{attribute 'linkalways'} 
{attribute 'no_explicit_call' := 'This FB is a CLASS and must be accessed using methods or properties'}
{attribute 'enable_dynamic_creation'}
FUNCTION_BLOCK Node_F_VN_BitwiseAndImages EXTENDS VisionNode
VAR
    ipSrcImage1 : _ITcVnImage;
    ipSrcImage2 : _ITcVnImage;
    ipDestImage : _ITcVnImage;
    hrPrev : _HRESULT(S_OK);
	hresult : _HRESULT(S_OK);
END_VAR

METHOD PUBLIC  Clone : I_Node
VAR
	pNode : POINTER TO Node_F_VN_BitwiseAndImages;
END_VAR
pNode := __NEW(Node_F_VN_BitwiseAndImages);
Clone := pNode^;
END_METHOD

METHOD FB_init : BOOL
VAR_INPUT
	bInitRetains : BOOL; // if TRUE, the retain variables are initialized (warm start / cold start)
	bInCopyCode : BOOL;  // if TRUE, the instance afterwards gets moved into the copy code (online change)
END_VAR
AddInput('ipSrcImage1', ipSrcImage1);
AddInput('ipSrcImage2', ipSrcImage2);
AddInput('hrPrev', hrPrev);
AddOutput('ipDestImage', ipDestImage);
AddOutput('hresult',hresult);
END_METHOD

METHOD PROTECTED OnExecute : HRESULT
hresult.Value := F_VN_BitwiseAndImages(
    ipSrcImage1 := ipSrcImage1.Value,
    ipSrcImage2 := ipSrcImage2.Value,
	ipDestImage := ipDestImage.Value,
	hrPrev:= hrPrev.Value);
END_METHOD

METHOD PUBLIC PreExecutionCheck
VAR_INPUT
	Check : I_PreExecutionChecks;
END_VAR
IF FAILED(hrPrev.Value) THEN
    RETURN;
END_IF

Check.IsTrue(ipSrcImage1.IsValid, 'ipSrcImage1 must contain an image');
Check.IsTrue(ipSrcImage2.IsValid, 'ipSrcImage2 must contain an image');
END_METHOD

END_FUNCTION_BLOCK

(* stored: Version 1.1.0.1, ProductVersion 3.1.4024.13
   POU Node_F_VN_BitwiseAndImages: Id {5576663e-5e63-02a7-00a4-3fe8d884f1a5}, SpecialFunc None
   Folder Constructor: Id {993ed1dd-331f-0909-1531-be08c12660e1}
   Method Clone: Id {53aa05c1-b5c6-0c2c-3180-39282481cded}
   Method FB_init: Id {4075234d-9032-0c1c-0d42-97d23e29d12c}
   Method OnExecute: Id {67e5e44a-bfed-0ead-082c-abacc700ab27}
   Method PreExecutionCheck: Id {29890d40-8d28-0320-1b83-acbb56324c2c} *)
